Staubli VAL3: onEnterEvent.pgx

program onEnterEvent()
begin
  //
  // Change the frame coordinate
  //
  if nFrame>0
    call page_changeTrsf(saveData:fFrameItem[nFrame].fFrame.trsf,false,false,sEvent,"")
  endIf
end
